Staubli VAL3: listcursor.pgx

public program listcursor(num pView (dimensions=1), bool pShow (dimensions=1))
  local num lX
  local num lY
  local string message
  local bool l_bEmpty
begin
  //
  // toneage Staubli Copyright 2005
  //
  call isListEmpty(l_bEmpty)
  if !l_bEmpty
    nView=pView
    lX=nTopX+1
    lY=nTopY+1+pView
    if (nView+nFirst)>(size(sItems)-1)
      call strfill(sItems[size(sItems)-1],nBottomX,message)
    else
      call strfill(sItems[nView+nFirst],nBottomX,message)
    endIf
    gotoxy(lX,lY)
    if (pShow==true)
      setTextMode(1)
      put(message)
      setTextMode(0)
    else
      setTextMode(0)
      put(message)
    endIf
  endIf
end
